// TwinCAT 3 PLC project PLC1
// ProgramVersion: 3.1.4020.4
// libraries:
//   Tc2_MC2, * (Beckhoff Automation GmbH)
//   Tc2_Standard, * (Beckhoff Automation GmbH)
//   Tc2_System, * (Beckhoff Automation GmbH)
//   Tc3_Module, * (Beckhoff Automation GmbH)
// project tree:
//   DataType/ MoveState_t.TcDUT (not stored)
//   / PlcTask.TcTTO
//   POUs/ AxisCtrl.TcPOU, MAIN.TcPOU (not stored)
// real-time tasks:
//   TASK PlcTask: cycle T#10ms, priority 20, ADS port 350
// motion (NC):
//   TASK NC-Task 1 SAF: cycle T#2ms, priority 4, ADS port 501
//   TASK NC-Task 1 SVB: cycle T#10ms, priority 8, ADS port 511
//   AXIS Axis 1 (id 1)
//     Dynamic: AccelerationMaximum=20000, DecelerationMaximum=20000, Acceleration=10000, Deceleration=10000, Jerk=219069
//     Velo: Maximum=1000
//     OtherSettings: AllowMotionCmdToSlave=true
//     encoder EncType=1
//       EncPara: ScaleFactorNumerator=90, ScaleFactorDenominator=65536
//         SoftEndMinControl: Range=100
//         SoftEndMaxControl: Range=900
//         Inc: RefSearchInverse=true
//     drive DrvType=5
//       Analog: VeloReferenz=1100
//       TimeComp: TaskDelayCycles=1
//     controller CtrType=1
//       CtrPara: PriorControlFactor=1
//         Observer: BandWidth=20
//   AXIS Axis 2 (id 2)
//     Dynamic: AccelerationMaximum=20000, DecelerationMaximum=20000, Acceleration=10000, Deceleration=10000, Jerk=219069
//     Velo: Maximum=1000
//     OtherSettings: AllowMotionCmdToSlave=true
//     encoder EncType=1
//       EncPara: ScaleFactorNumerator=90, ScaleFactorDenominator=65536
//         SoftEndMinControl: Range=100
//         SoftEndMaxControl: Range=900
//         Inc: RefSearchInverse=true
//     drive DrvType=5
//       Analog: VeloReferenz=1100
//       TimeComp: TaskDelayCycles=1
//     controller CtrType=1
//       CtrPara: PriorControlFactor=1
//         Observer: BandWidth=20
//   AXIS Axis 3 (id 3)
//     Dynamic: AccelerationMaximum=20000, DecelerationMaximum=20000, Acceleration=10000, Deceleration=10000, Jerk=219069
//     Velo: Maximum=1000
//     OtherSettings: AllowMotionCmdToSlave=true
//     encoder EncType=1
//       EncPara: ScaleFactorNumerator=90, ScaleFactorDenominator=65536
//         SoftEndMinControl: Range=100
//         SoftEndMaxControl: Range=900
//         Inc: RefSearchInverse=true
//     drive DrvType=5
//       Analog: VeloReferenz=1100
//       TimeComp: TaskDelayCycles=1
//     controller CtrType=1
//       CtrPara: PriorControlFactor=1
//         Observer: BandWidth=20
//   AXIS Axis 4 (id 4)
//     Dynamic: AccelerationMaximum=20000, DecelerationMaximum=20000, Acceleration=10000, Deceleration=10000, Jerk=219069
//     Velo: Maximum=1000
//     OtherSettings: AllowMotionCmdToSlave=true
//     encoder EncType=1
//       EncPara: ScaleFactorNumerator=90, ScaleFactorDenominator=65536
//         SoftEndMinControl: Range=100
//         SoftEndMaxControl: Range=900
//         Inc: RefSearchInverse=true
//     drive DrvType=5
//       Analog: VeloReferenz=1100
//       TimeComp: TaskDelayCycles=1
//     controller CtrType=1
//       CtrPara: PriorControlFactor=1
//         Observer: BandWidth=20
//   AXIS Axis 5 (id 5)
//     Dynamic: AccelerationMaximum=20000, DecelerationMaximum=20000, Acceleration=10000, Deceleration=10000, Jerk=219069
//     Velo: Maximum=1000
//     OtherSettings: AllowMotionCmdToSlave=true
//     encoder EncType=1
//       EncPara: ScaleFactorNumerator=90, ScaleFactorDenominator=65536
//         SoftEndMinControl: Range=100
//         SoftEndMaxControl: Range=900
//         Inc: RefSearchInverse=true
//     drive DrvType=5
//       Analog: VeloReferenz=1100
//       TimeComp: TaskDelayCycles=1
//     controller CtrType=1
//       CtrPara: PriorControlFactor=1
//         Observer: BandWidth=20
//   AXIS Axis 6 (id 6)
//     Dynamic: AccelerationMaximum=20000, DecelerationMaximum=20000, Acceleration=10000, Deceleration=10000, Jerk=219069
//     Velo: Maximum=1000
//     OtherSettings: AllowMotionCmdToSlave=true
//     encoder EncType=1
//       EncPara: ScaleFactorNumerator=90, ScaleFactorDenominator=65536
//         SoftEndMinControl: Range=100
//         SoftEndMaxControl: Range=900
//         Inc: RefSearchInverse=true
//     drive DrvType=5
//       Analog: VeloReferenz=1100
//       TimeComp: TaskDelayCycles=1
//     controller CtrType=1
//       CtrPara: PriorControlFactor=1
//         Observer: BandWidth=20
//   AXIS Axis 7 (id 7)
//     Dynamic: AccelerationMaximum=20000, DecelerationMaximum=20000, Acceleration=10000, Deceleration=10000, Jerk=219069
//     Velo: Maximum=1000
//     OtherSettings: AllowMotionCmdToSlave=true
//     encoder EncType=1
//       EncPara: ScaleFactorNumerator=90, ScaleFactorDenominator=65536
//         SoftEndMinControl: Range=100
//         SoftEndMaxControl: Range=900
//         Inc: RefSearchInverse=true
//     drive DrvType=5
//       Analog: VeloReferenz=1100
//       TimeComp: TaskDelayCycles=1
//     controller CtrType=1
//       CtrPara: PriorControlFactor=1
//         Observer: BandWidth=20
//   AXIS Axis 8 (id 8)
//     Dynamic: AccelerationMaximum=20000, DecelerationMaximum=20000, Acceleration=10000, Deceleration=10000, Jerk=219069
//     Velo: Maximum=1000
//     OtherSettings: AllowMotionCmdToSlave=true
//     encoder EncType=1
//       EncPara: ScaleFactorNumerator=90, ScaleFactorDenominator=65536
//         SoftEndMinControl: Range=100
//         SoftEndMaxControl: Range=900
//         Inc: RefSearchInverse=true
//     drive DrvType=5
//       Analog: VeloReferenz=1100
//       TimeComp: TaskDelayCycles=1
//     controller CtrType=1
//       CtrPara: PriorControlFactor=1
//         Observer: BandWidth=20
//   AXIS Axis 9 (id 9)
//     Dynamic: AccelerationMaximum=20000, DecelerationMaximum=20000, Acceleration=10000, Deceleration=10000, Jerk=219069
//     Velo: Maximum=1000
//     OtherSettings: AllowMotionCmdToSlave=true
//     encoder EncType=1
//       EncPara: ScaleFactorNumerator=90, ScaleFactorDenominator=65536
//         SoftEndMinControl: Range=100
//         SoftEndMaxControl: Range=900
//         Inc: RefSearchInverse=true
//     drive DrvType=5
//       Analog: VeloReferenz=1100
//       TimeComp: TaskDelayCycles=1
//     controller CtrType=1
//       CtrPara: PriorControlFactor=1
//         Observer: BandWidth=20
//   AXIS Axis 10 (id 10)
//     Dynamic: AccelerationMaximum=20000, DecelerationMaximum=20000, Acceleration=10000, Deceleration=10000, Jerk=219069
//     Velo: Maximum=1000
//     OtherSettings: AllowMotionCmdToSlave=true
//     encoder EncType=1
//       EncPara: ScaleFactorNumerator=90, ScaleFactorDenominator=65536
//         SoftEndMinControl: Range=100
//         SoftEndMaxControl: Range=900
//         Inc: RefSearchInverse=true
//     drive DrvType=5
//       Analog: VeloReferenz=1100
//       TimeComp: TaskDelayCycles=1
//     controller CtrType=1
//       CtrPara: PriorControlFactor=1
//         Observer: BandWidth=20
// I/O:
//   DEVICE NIC (disabled), AmsNetId 192.168.2.43.2.1
//     Ctr1 [CMMP-AS V4p0 CiA402]
//     Ctr2 [CMMP-AS V4p0 CiA402]
// variable links:
//   NC-Task 1 SAF/Axes/Axis 2 <-> NIC/Ctr1
//     Enc/Inputs/In/nDataIn1 <-> Inputs/Position_Actual_Value
//     Enc/Inputs/In/nDcInputTime <-> InfoData/DcInputShift
//     Enc/Inputs/In/nState4 @bit 1 <-> WcState/InputToggle
//     Enc/Inputs/In/nState4 <-> WcState/WcState
//   PLC1/PLC1 Instance <-> NC-Task 1 SAF/Axes/Axis 1
//     PlcTask Inputs/MAIN.axisCtrls[1].axis.NcToPlc <-> Outputs/ToPlc
//     PlcTask Outputs/MAIN.axisCtrls[1].axis.PlcToNc <-> Inputs/FromPlc
//   PLC1/PLC1 Instance <-> NC-Task 1 SAF/Axes/Axis 10
//     PlcTask Inputs/MAIN.axisCtrls[10].axis.NcToPlc <-> Outputs/ToPlc
//     PlcTask Outputs/MAIN.axisCtrls[10].axis.PlcToNc <-> Inputs/FromPlc
//   PLC1/PLC1 Instance <-> NC-Task 1 SAF/Axes/Axis 2
//     PlcTask Inputs/MAIN.axisCtrls[2].axis.NcToPlc <-> Outputs/ToPlc
//     PlcTask Outputs/MAIN.axisCtrls[2].axis.PlcToNc <-> Inputs/FromPlc
//   PLC1/PLC1 Instance <-> NC-Task 1 SAF/Axes/Axis 3
//     PlcTask Inputs/MAIN.axisCtrls[3].axis.NcToPlc <-> Outputs/ToPlc
//     PlcTask Outputs/MAIN.axisCtrls[3].axis.PlcToNc <-> Inputs/FromPlc
//   PLC1/PLC1 Instance <-> NC-Task 1 SAF/Axes/Axis 4
//     PlcTask Inputs/MAIN.axisCtrls[4].axis.NcToPlc <-> Outputs/ToPlc
//     PlcTask Outputs/MAIN.axisCtrls[4].axis.PlcToNc <-> Inputs/FromPlc
//   PLC1/PLC1 Instance <-> NC-Task 1 SAF/Axes/Axis 5
//     PlcTask Inputs/MAIN.axisCtrls[5].axis.NcToPlc <-> Outputs/ToPlc
//     PlcTask Outputs/MAIN.axisCtrls[5].axis.PlcToNc <-> Inputs/FromPlc
//   PLC1/PLC1 Instance <-> NC-Task 1 SAF/Axes/Axis 6
//     PlcTask Inputs/MAIN.axisCtrls[6].axis.NcToPlc <-> Outputs/ToPlc
//     PlcTask Outputs/MAIN.axisCtrls[6].axis.PlcToNc <-> Inputs/FromPlc
//   PLC1/PLC1 Instance <-> NC-Task 1 SAF/Axes/Axis 7
//     PlcTask Inputs/MAIN.axisCtrls[7].axis.NcToPlc <-> Outputs/ToPlc
//     PlcTask Outputs/MAIN.axisCtrls[7].axis.PlcToNc <-> Inputs/FromPlc
//   PLC1/PLC1 Instance <-> NC-Task 1 SAF/Axes/Axis 8
//     PlcTask Inputs/MAIN.axisCtrls[8].axis.NcToPlc <-> Outputs/ToPlc
//     PlcTask Outputs/MAIN.axisCtrls[8].axis.PlcToNc <-> Inputs/FromPlc
//   PLC1/PLC1 Instance <-> NC-Task 1 SAF/Axes/Axis 9
//     PlcTask Inputs/MAIN.axisCtrls[9].axis.NcToPlc <-> Outputs/ToPlc
//     PlcTask Outputs/MAIN.axisCtrls[9].axis.PlcToNc <-> Inputs/FromPlc

CONFIGURATION PLC1
    RESOURCE PLC ON TwinCAT3
        TASK PlcTask(INTERVAL := T#10ms, PRIORITY := 20);
        PROGRAM MAIN WITH PlcTask : MAIN;
    END_RESOURCE
END_CONFIGURATION

// ---- POUs/AxisCtrl.TcPOU
FUNCTION_BLOCK AxisCtrl
VAR_INPUT
END_VAR
VAR_OUTPUT
END_VAR
VAR
	axis : AXIS_REF;
	state : MoveState_t;
	
	moveAbs: MC_MoveAbsolute;
	moveAbsOut: ST_McOutputs;

	power: MC_Power;
	powerOut : ST_McOutputs;
	
	reset: MC_Reset;
	resetOut : ST_McOutputs;
	
	cmd_pos : LREAL;
	cmd_vel : LREAL;
	cmd_acc : LREAL;
	cmd_vel_end : LREAL;
	cmd_need_exe : BOOL;
	
	readActPos: MC_ReadActualPosition;
	readActVel: MC_ReadActualVelocity;
	
	actPosOut : ST_McOutputs;
	actVelOut : ST_McOutputs;
	
	actual_pos : LREAL;
	actual_vel : LREAL;
END_VAR

	axis.ReadStatus();
	
	CASE state OF
		
		MOVESTATE_INIT :
			moveAbs.Execute := FALSE;
			reset.Execute := FALSE;
			power.Enable := FALSE;
			
		MOVESTATE_ENABLE:
			power.Enable := TRUE;

			IF power.Error THEN
				state := MOVESTATE_ERROR;
			ELSE
				state := MOVESTATE_MOVING;
			END_IF
		
		MOVESTATE_HOMING:
			state := MOVESTATE_MOVING;
		
		MOVESTATE_MOVING:		
			IF cmd_need_exe THEN
				moveAbs.Position := cmd_pos;
				moveAbs.Velocity := cmd_vel;
				moveAbs.BufferMode := MC_Buffered;
				moveAbs.Execute := TRUE;
				cmd_need_exe := FALSE;			
			END_IF;		
		
			IF moveAbs.Done THEN
				moveAbs.Execute := FALSE;
			ELSIF moveAbs.CommandAborted OR moveAbs.Error THEN
				state := MOVESTATE_ERROR;
			END_IF
			
		MOVESTATE_ERROR :
			IF axis.Status.Error THEN
				state := MOVESTATE_RESET;
			ELSE
				state := MOVESTATE_INIT;
			END_IF

		MOVESTATE_RESET :
			reset.Execute := TRUE;
			IF reset.Done THEN
				state := MOVESTATE_INIT;
			ELSIF reset.Error THEN
				state := MOVESTATE_INIT;
			END_IF
	END_CASE
	
	
	ActPower();
	ActMove();
	ActReset();
	ActRead();

ACTION ActMove:
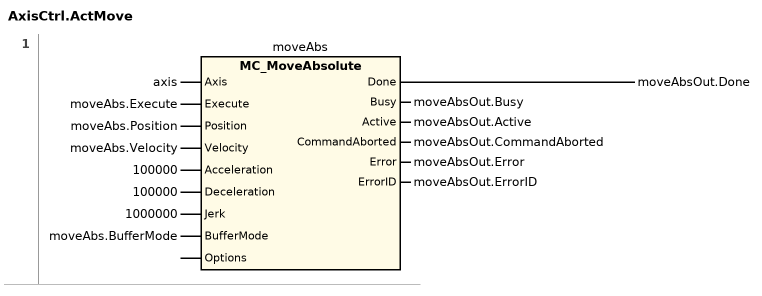
// NETWORK 1
moveAbs(
    Axis := axis,
    Execute := moveAbs.Execute,
    Position := moveAbs.Position,
    Velocity := moveAbs.Velocity,
    Acceleration := 100000,
    Deceleration := 100000,
    Jerk := 1000000,
    BufferMode := moveAbs.BufferMode,
    Busy => moveAbsOut.Busy,
    Active => moveAbsOut.Active,
    CommandAborted => moveAbsOut.CommandAborted,
    Error => moveAbsOut.Error,
    ErrorID => moveAbsOut.ErrorID); // MC_MoveAbsolute
moveAbsOut.Done := moveAbs.Done;
END_ACTION

ACTION ActPower:
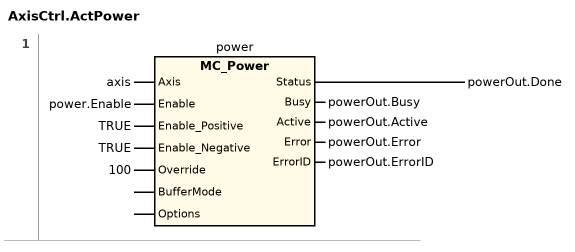
// NETWORK 1
power(
    Axis := axis,
    Enable := power.Enable,
    Enable_Positive := TRUE,
    Enable_Negative := TRUE,
    Override := 100,
    Busy => powerOut.Busy,
    Active => powerOut.Active,
    Error => powerOut.Error,
    ErrorID => powerOut.ErrorID); // MC_Power
powerOut.Done := power.Status;
END_ACTION

ACTION ActRead:
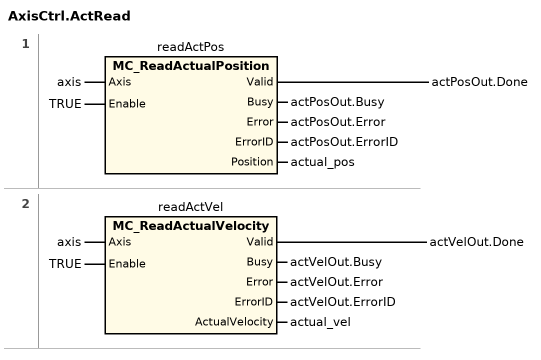
// NETWORK 1
readActPos(
    Axis := axis,
    Enable := TRUE,
    Busy => actPosOut.Busy,
    Error => actPosOut.Error,
    ErrorID => actPosOut.ErrorID,
    Position => actual_pos); // MC_ReadActualPosition
actPosOut.Done := readActPos.Valid;

// NETWORK 2
readActVel(
    Axis := axis,
    Enable := TRUE,
    Busy => actVelOut.Busy,
    Error => actVelOut.Error,
    ErrorID => actVelOut.ErrorID,
    ActualVelocity => actual_vel); // MC_ReadActualVelocity
actVelOut.Done := readActVel.Valid;
END_ACTION

ACTION ActReset:
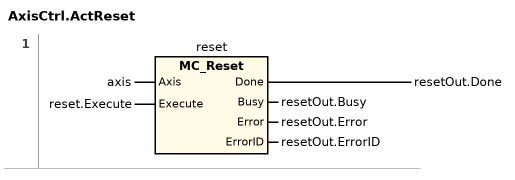
// NETWORK 1
reset(
    Axis := axis,
    Execute := reset.Execute,
    Busy => resetOut.Busy,
    Error => resetOut.Error,
    ErrorID => resetOut.ErrorID); // MC_Reset
resetOut.Done := reset.Done;
END_ACTION

END_FUNCTION_BLOCK
